FUNCTION_BLOCK FB_5_TransferirBase_SFC
VAR_INPUT
	
	//  SFC-Flags
	SFCPause: BOOL;
	SFCReset: BOOL;

	// Indicadores de sincronización
	Ack: BOOL := TRUE;
	Execute: BOOL;
	
	// Entradas
	PalePresencia: BOOL;
	
END_VAR
VAR_OUTPUT
	
	// Indicadores de sincronización
	Ready: BOOL;	
	Done: BOOL;
	
	// Salidas
	CintaMotorActiva: BOOL;
	CintaRetenedorBaja: BOOL;
	CintaSeparadorSube: BOOL;
	
END_VAR
VAR
END_VAR

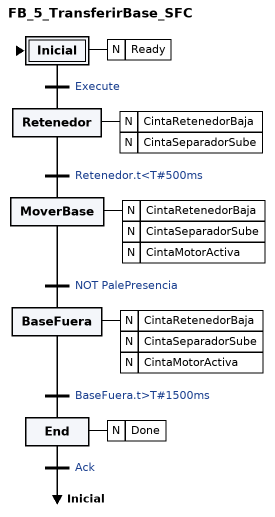
INITIAL_STEP Inicial:
    Ready(N);
END_STEP
TRANSITION FROM Inicial TO Retenedor
    := Execute;
END_TRANSITION
STEP Retenedor:
    CintaRetenedorBaja(N);
    CintaSeparadorSube(N);
END_STEP
TRANSITION FROM Retenedor TO MoverBase
    := Retenedor.t<T#500ms;
END_TRANSITION
STEP MoverBase:
    CintaRetenedorBaja(N);
    CintaSeparadorSube(N);
    CintaMotorActiva(N);
END_STEP
TRANSITION FROM MoverBase TO BaseFuera
    := NOT PalePresencia;
END_TRANSITION
STEP BaseFuera:
    CintaRetenedorBaja(N);
    CintaSeparadorSube(N);
    CintaMotorActiva(N);
END_STEP
TRANSITION FROM BaseFuera TO End
    := BaseFuera.t>T#1500ms;
END_TRANSITION
STEP End:
    Done(N);
END_STEP
TRANSITION FROM End TO Inicial
    := Ack;
END_TRANSITION

END_FUNCTION_BLOCK

(* stored: Version 1.1.0.1, ProductVersion 3.1.4024.12
   POU FB_5_TransferirBase_SFC: Id {b439ffa1-ca82-4ec3-9751-cbfe00d05d8d}, SpecialFunc None *)
